(* IEC 61131-3 sources: Lasal/CPU_5344_V01/Class/Invert, 1 file *)

(* ---- Invert.st ---- *)
(*!
<Class
	Name               = "Invert"
	Revision           = "0.0"
	RealtimeTask       = "false"
	CyclicTask         = "false"
	BackgroundTask     = "false"
	Sigmatek           = "false"
	OSInterface        = "false"
	HighPriority       = "false"
	Automatic          = "false"
	UpdateMode         = "Prescan"
	SharedCommandTable = "true"
	Objectsize         = "(300,180)">
	<Channels>
		<Server Name="ClassSvr" Visualized="false" Initialize="false" WriteProtected="true" Retentive="false"/>
		<Server Name="InvertUit" Visualized="false" Initialize="false" WriteProtected="false" Retentive="SRam"/>
		<Client Name="Client" Required="true" Internal="false"/>
	</Channels>
</Class>
*)
Invert : CLASS
  //Servers:
	ClassSvr 	: SvrChCmd_DINT;
	InvertUit 	: SvrCh_DINT;
  //Clients:
	Client 	: CltCh_DINT;
  //Variables:
  //Functions:

	FUNCTION VIRTUAL GLOBAL ClassSvr::Read
		VAR_OUTPUT
			output (EAX) 	: DINT;
		END_VAR;
  //Tables:
	FUNCTION @STD
		VAR_OUTPUT
			ret_code	: CONFSTATES;
		END_VAR;
	FUNCTION GLOBAL TAB @CT_;
END_CLASS;

FUNCTION VIRTUAL GLOBAL Invert::ClassSvr::Read
	VAR_OUTPUT
		output (EAX) 	: DINT;
	END_VAR
  Client := Client.Read();
  if InvertUit = 0 then
    if Client = 1 then
      ClassSvr := 0;
    else
      ClassSvr := 1;
    end_if;
  else
    ClassSvr := Client;
  end_if;
	output := ClassSvr;

END_FUNCTION
